(* IEC 61131-3 sources: Industry-PLC-LLM/data/PLCBEAD_repo/PLCBEAD_PLCEmbed-main/PLC-BEAD/Source/GEB/BIT_LOAD_DW2, 1 file *)

(* ---- BIT_LOAD_DW2.ST ---- *)
FUNCTION BIT_LOAD_DW2:DWORD
	VAR_INPUT
		I :	DWORD;
		D :	BOOL;
		P :	INT;
		N :	INT;
	END_VAR

	IF D THEN
		BIT_LOAD_DW2 := ROL(SHR(DWORD#16#FFFFFFFF, 32 - N) OR ROR(I, P), P);
	ELSE
		BIT_LOAD_DW2 := ROL(SHL(DWORD#16#FFFFFFFF, N) AND ROR(I, P), P);
	END_IF;

END_FUNCTION

PROGRAM program0
  VAR
    LocalVar0 : DWORD;
	LocalVaR1  : BOOL;
	LocalVaR2 : INT;
	LocalVar3 : INT;
    LocalOUT  : DWORD;
  END_VAR

  LocalOUT := BIT_LOAD_DW2(LocalVar0, LocalVaR1 , LocalVaR2, LocalVar3);
END_PROGRAM
